// TIA Portal V18 export
TYPE "RTD"
// stored: IsFailsafeCompliant false
   STRUCT
      "RECUPERATION TANK" : Int;
      "HOT WATER TANK" : Int;
      "CAUSTIC TANK" : Int;
      "ACID TANK" : Int;
      "FWD LINE" : Int;
      "RETURN LINE" : Int;
      "SPARE RTD" : Int;
      "SPARE RTD 1" : Int;
   END_STRUCT;
END_TYPE
